_fbResult.P_MethodResult := ap_fbEventsExecute[0]^.M_Execute(_fbResult.P_MethodResult);
END_METHOD

METHOD PUBLIC M_ExecuteControl : HResult //needs to run all the time
VAR_INPUT
END_VAR
VAR
	loopCounter : DINT;
	currentState : E_PackMLStates;
END_VAR
_mapping();
currentState := state;
FOR loopCounter := 0 TO 20 BY 1 DO 
	CASE state OF
		E_PackMLStates.aborted:
			M_Aborted();
		E_PackMLStates.aborting:
			M_Aborting();
		E_PackMLStates.complete:
			stateMachineResult := M_Complete(stateMachineResult);
			IF stateMachineResult = MPM_FBResult.E_Result.S_OK THEN
				state := E_PackMLStates.complete;
			END_IF		
		E_PackMLStates.completing:	
			stateMachineResult := M_Completing(stateMachineResult);
			IF stateMachineResult = MPM_FBResult.E_Result.S_OK THEN
				state := E_PackMLStates.idle;
			END_IF					
		E_PackMLStates.execute:	
			stateMachineResult := M_Execute(stateMachineResult);	
			IF stateMachineResult = MPM_FBResult.E_Result.S_OK THEN
				state := E_PackMLStates.completing;
			END_IF			
		E_PackMLStates.held:	
			M_Held();	
		E_PackMLStates.holding:	
			M_Holding();		
		E_PackMLStates.idle:	
			stateMachineResult := M_Idle(stateMachineResult);		
			IF stateMachineResult = MPM_FBResult.E_Result.S_WORKING AND start = TRUE THEN
				stateMachineResult := MPM_FBResult.E_Result.S_OK;
				start := FALSE;
				state := E_PackMLStates.starting;
			END_IF	
		E_PackMLStates.starting:	
			stateMachineResult := M_Starting(stateMachineResult);
			IF stateMachineResult = MPM_FBResult.E_Result.S_OK THEN
				state := E_PackMLStates.execute;
			END_IF		
		E_PackMLStates.stopped:	
			M_Stopped();	
		E_PackMLStates.stopping:	
			M_Stopping();
		E_PackMLStates.suspdending:	
			M_Suspending();		
		E_PackMLStates.suspended:	
			M_Suspended();	
		E_PackMLStates.un_holding:	
			M_Un_Holding();			
		E_PackMLStates.un_suspsending:	
			M_Un_Suspending();					
	END_CASE
	
	IF currentState = state THEN // if state didnt change
	 	EXIT;
	ELSE // if state changed
		currentState := state;
	END_IF
	
END_FOR
END_METHOD

METHOD PUBLIC M_Held : HResult
VAR_INPUT
END_VAR
VAR_OUTPUT
	abort : BOOL;
	stop : BOOL;
END_VAR
END_METHOD

METHOD PUBLIC M_Holding : HResult
VAR_INPUT
END_VAR
VAR_OUTPUT
	abort : BOOL;
	stop : BOOL;
END_VAR
END_METHOD

METHOD PUBLIC M_Idle : HResult
VAR_INPUT
	lastResult : HResult;
END_VAR
VAR_OUTPUT
	abort : BOOL;
END_VAR
VAR_INST
	_fbResult : FB_ResultHelper_V2_1;	
	_lastResult : HRESULT;
	_state : POINTER TO DINT;
END_VAR
_state := ADR(state_idle);
IF _fbResult.M_MethodResult(M_Idle,lastResult,ADR(_lastResult)) = FALSE THEN
	RETURN;
END_IF

_fbResult.P_MethodResult := ap_fbEventsIdle[0]^.M_Execute(_fbResult.P_MethodResult);
END_METHOD

METHOD PUBLIC M_Resetting : HResult
VAR_INPUT
END_VAR
VAR_OUTPUT
	abort : BOOL;
	stop : BOOL;
END_VAR
END_METHOD

METHOD M_Starting : HResult
VAR_INPUT
	lastResult : HResult;
END_VAR
VAR_OUTPUT
	abort : BOOL;
END_VAR
VAR_INST
	_fbResult : FB_ResultHelper_V2_1;	
	_lastResult : HRESULT;
	_state : POINTER TO DINT;
END_VAR
_state := ADR(state_starting);
IF _fbResult.M_MethodResult(M_Starting,lastResult,ADR(_lastResult)) = FALSE THEN
	RETURN;
END_IF

IF _fbResult.P_MethodResult = E_Result.S_OK THEN
	_state^ := 0;
END_IF

_fbResult.P_MethodResult := ap_fbEventsStarting[0]^.M_Execute(_fbResult.P_MethodResult);
END_METHOD

METHOD PUBLIC M_Stopped : HResult
VAR_INPUT
	
END_VAR
VAR_OUTPUT
	abort : BOOL;
END_VAR
END_METHOD

METHOD PUBLIC M_Stopping : HResult
VAR_INPUT
END_VAR
VAR_OUTPUT
	abort : BOOL;
END_VAR
END_METHOD

METHOD PUBLIC M_Suspended : HREsult
VAR_INPUT
END_VAR
VAR_OUTPUT
	abort : BOOL;
	stop : BOOL;
END_VAR
END_METHOD

METHOD PUBLIC M_Suspending : HREsult
VAR_INPUT
END_VAR
VAR_OUTPUT
	abort : BOOL;
	stop : BOOL;
END_VAR
END_METHOD

METHOD PUBLIC M_Un_Holding : HREsult
VAR_INPUT
END_VAR
VAR_OUTPUT
	abort : BOOL;
	stop : BOOL;
END_VAR
END_METHOD

METHOD PUBLIC M_Un_Suspending : HREsult
VAR_INPUT
END_VAR
VAR_OUTPUT
	abort : BOOL;
	stop : BOOL;
END_VAR
END_METHOD

END_FUNCTION_BLOCK

// ---- FBs/Abstracts/FB_PackMLControl.TcPOU
(*
Standard way to control assests in system
*)
FUNCTION_BLOCK ABSTRACT FB_PackMLControl
VAR_INPUT
END_VAR
VAR_OUTPUT
END_VAR
VAR
	state_idle : DINT;
	state_starting : DINT;
	state_execute : DINT;	
	state_completing : DINT;			
	state_complete : DINT;		
	start : BOOL;
	complete : BOOL;
	stateMachineResult : HResult;
	packMLStop : BOOL;
END_VAR

METHOD PUBLIC ABSTRACT M_Aborted : HResult
VAR_INPUT
END_VAR
END_METHOD

METHOD PUBLIC ABSTRACT M_Aborting : HResult
VAR_INPUT
END_VAR
END_METHOD

METHOD PUBLIC ABSTRACT M_Complete : HResult
VAR_INPUT
	lastResult : HResult;
END_VAR
VAR_OUTPUT
	abort : BOOL;
END_VAR
END_METHOD

METHOD PUBLIC ABSTRACT M_Completing : HREsult
VAR_INPUT
	lastResult : HResult;
END_VAR
VAR_OUTPUT
	abort : BOOL;	
	stop : BOOL;
END_VAR
END_METHOD

METHOD PUBLIC ABSTRACT M_Execute : HResult
VAR_INPUT
	lastResult : HResult;
END_VAR
VAR_OUTPUT
	stop : BOOL;
	suspend : BOOL;
	hold : BOOL;
END_VAR
END_METHOD

METHOD PUBLIC ABSTRACT M_Held : HResult
VAR_INPUT
END_VAR
VAR_OUTPUT
	abort : BOOL;
	stop : BOOL;
END_VAR
END_METHOD

METHOD PUBLIC ABSTRACT M_Holding : HResult
VAR_INPUT
END_VAR
VAR_OUTPUT
	abort : BOOL;
	stop : BOOL;
END_VAR
END_METHOD

METHOD PUBLIC ABSTRACT M_Idle : HResult
VAR_INPUT
	lastResult : HResult;
END_VAR
VAR_OUTPUT
	abort : BOOL;
END_VAR
END_METHOD

METHOD PUBLIC ABSTRACT M_Resetting : HResult
VAR_INPUT
END_VAR
VAR_OUTPUT
	abort : BOOL;
	stop : BOOL;
END_VAR
END_METHOD

METHOD ABSTRACT M_Starting : HResult
VAR_INPUT
	lastResult : HResult;
END_VAR
VAR_OUTPUT
	abort : BOOL;
END_VAR
END_METHOD

METHOD PUBLIC ABSTRACT M_Stopped : HResult
VAR_INPUT
END_VAR
VAR_OUTPUT
	abort : BOOL;
END_VAR
END_METHOD

METHOD PUBLIC ABSTRACT M_Stopping : HResult
VAR_INPUT
END_VAR
VAR_OUTPUT
	abort : BOOL;
END_VAR
END_METHOD

METHOD PUBLIC ABSTRACT M_Suspended : HREsult
VAR_INPUT
END_VAR
VAR_OUTPUT
	abort : BOOL;
	stop : BOOL;
END_VAR
END_METHOD

METHOD PUBLIC ABSTRACT M_Suspending : HREsult
VAR_INPUT
END_VAR
VAR_OUTPUT
	abort : BOOL;
	stop : BOOL;
END_VAR
END_METHOD

METHOD PUBLIC ABSTRACT M_Un_Holding : HREsult
VAR_INPUT
END_VAR
VAR_OUTPUT
	abort : BOOL;
	stop : BOOL;
END_VAR
END_METHOD

METHOD PUBLIC ABSTRACT M_Un_Suspending : HREsult
VAR_INPUT
END_VAR
VAR_OUTPUT
	abort : BOOL;
	stop : BOOL;
END_VAR
END_METHOD

END_FUNCTION_BLOCK

// ---- FBs/FB_Kinenmatics.TcPOU
FUNCTION_BLOCK FB_Kinenmatics
VAR_INPUT
	intialVelocity : LREAL;
	jerkLimit : LREAL;
	accelLimit : LREAL;
	decelLimit : LREAL;
	velocityLimit : LREAL;
	positionDelta : LREAL;
	timeToComplete : LREAL;
	discriment : LREAL;
END_VAR
VAR_OUTPUT
	minTime : LREAL;
	velocityOutput : LREAL;
	accelOutput : LREAL;
	jerkOutput : LREAL;
	error : BOOL;
	errorMsg : STRING;	
END_VAR
VAR
	positionMid : LREAL;
	positionQuarter : LREAL;
	//Caculating max values for a Jerk limited move
	jerkMoveAccelMax : LREAL;
	jerkMoveTimeToMaxAccel : LREAL;
	jerkMoveVelocityAtMaxAccel : LREAL;	
	jerkMoveVelocityMax : LREAL;
	jerkMoveTimeToMaxVelocity : LREAL;
	jerkMoveTimeToCompleteMin : LREAL;
	jerkMoveJerkLimitForTargetTime : LREAL;
	
	accelMoveTimeToMaxAccel : LREAL;
	accelMoveMaxVelocity : LREAL;
	accelMoveTimeForAccelConstantMove : LREAL;
	accelMoveTimeToCompleteMove : LREAL;

	accelMoveNewMaxAccel: LREAL;

	accelVelocityMoveTimeToMaxVelocity : LREAL;	
	accelVelocityMoveTimeFromMaxVelocityToMidPoint : LREAL;	
	accelVelocityTimeToCompleteMove : LREAL;
	accelSegment : ARRAY [0..6] OF LREAL;
	velocitySegment	: ARRAY [0..6] OF LREAL;
	positionSegment : ARRAY [0..6] OF LREAL;
	
	a : LREAL;
	b : LREAL;
	c : LREAL;
	


END_VAR

IF positionDelta <= 0 OR timeToComplete <= 0 OR accelLimit <= 0 OR decelLimit <= 0 OR velocityLimit <= 0 OR jerkLimit <= 0 THEN
	RETURN;
END_IF

positionMid := positionDelta/2.0;
positionQuarter := positionDelta/4.0;

//Solve for t jerk limited equation positionMid = jerkLimit * t^3, 
//t = (positionMid/jerkLimit) ^(1/3) where t = 1/4 of the time to complete the move
jerkMoveTimeToMaxAccel := EXPT(positionMid/jerkLimit,1.0/3.0);
jerkMoveAccelMax := jerkLimit * jerkMoveTimeToMaxAccel;
jerkMoveVelocityAtMaxAccel := jerkMoveTimeToMaxAccel * jerkMoveAccelMax;
jerkMoveTimeToCompleteMin := jerkMoveTimeToMaxAccel * 4.0;

IF jerkMoveTimeToCompleteMin > timeToComplete THEN
	minTime := jerkMoveTimeToCompleteMin;
	errorMsg := 'Jerk limit too low';
	error := TRUE;			
	RETURN;
ELSE
	errorMsg := '';	
	error := FALSE;			
END_IF

IF (accelLimit < jerkMoveAccelMax) OR velocityLimit <= jerkMoveVelocityAtMaxAccel THEN
	//Caculate known values
	accelMoveTimeToMaxAccel := accelLimit/jerkLimit;
	positionSegment[0] := 1.0/6.0 * jerkLimit * EXPT(accelMoveTimeToMaxAccel,3.0);
	velocitySegment[0] := 0.5 * jerkLimit * EXPT(accelMoveTimeToMaxAccel,2.0) + intialVelocity;
	accelSegment[0] := jerkLimit*accelMoveTimeToMaxAccel;
	
	//set up quardatic formula 
	// 1/2*accelLimit*t^2 + (velocitySegment[0] + (accelLimit[0]*accelMoveTimeToMaxAccel)*t + (velocitySegment[0] * accelMoveTimeToMaxAccel)+accelSegment[0]*0.5*accelMoveTimeToMaxAccel^2
	a := 0.5 * accelSegment[0];
	b :=  velocitySegment[0] + accelSegment[0]*accelMoveTimeToMaxAccel;
	c := ((velocitySegment[0] * accelMoveTimeToMaxAccel)+accelSegment[0]*0.5*EXPT(accelMoveTimeToMaxAccel,2.0)) - positionMid;
	
	//Make sure discriment > 0 otherwise program will crash
	discriment := (EXPT(b,2.0) - 4.0 * a *c);
	IF discriment > 0 THEN
		//caculate min time
		accelMoveTimeForAccelConstantMove := (-b + EXPT(EXPT(b,2.0) -4.0 * a *c,0.5))/(2*a); //solve for quadtratic
		accelMoveTimeToCompleteMove := 2.0*(accelMoveTimeToMaxAccel * 2.0 + accelMoveTimeForAccelConstantMove); // This value is the fastest the machine can move with the accel limit
		accelMoveMaxVelocity := accelMoveTimeToCompleteMove/2*accelSegment[0]-EXPT(accelSegment[0],2.0)/jerkLimit;
		//end of caculate min time
		IF accelMoveMaxVelocity > velocityLimit THEN
			accelVelocityMoveTimeToMaxVelocity := velocityLimit/accelLimit + accelLimit/(jerkLimit);
			positionSegment[1] := velocitySegment[0]*(accelVelocityMoveTimeToMaxVelocity-2.0*accelMoveTimeToMaxAccel) + 0.5*accelLimit*EXPT((accelVelocityMoveTimeToMaxVelocity-2.0*accelMoveTimeToMaxAccel),2.0);
			velocitySegment[1] := velocitySegment[0] + accelLimit * (accelVelocityMoveTimeToMaxVelocity-2.0*accelMoveTimeToMaxAccel);
			positionSegment[2] := velocitySegment[1] * accelMoveTimeToMaxAccel +  0.5*accelLimit*EXPT((accelMoveTimeToMaxAccel),2.0) - 1.0/6.0 * jerkLimit * EXPT(accelMoveTimeToMaxAccel,3.0);
			//positionSegment[0] :=velocitySegment[0]*(accelVelocityMoveTimeToMaxVelocity-2.0*accelMoveTimeToMaxAccel);
			positionSegment[3] := positionMid - (positionSegment[0] + positionSegment[1] + positionSegment[2]);
			accelVelocityMoveTimeFromMaxVelocityToMidPoint := positionSegment[3]/velocityLimit;
			accelVelocityTimeToCompleteMove := 2.0*(accelVelocityMoveTimeToMaxVelocity + accelVelocityMoveTimeFromMaxVelocityToMidPoint);
			IF	accelVelocityTimeToCompleteMove < timeToComplete THEN
				errorMsg := '';		
				error := FALSE;						
				a := 1/jerkLimit;
				b := -(accelVelocityMoveTimeToMaxVelocity + timeToComplete - accelVelocityTimeToCompleteMove); //-timeToComplete/2.0; //
				c := velocityLimit;
				discriment := (EXPT(b,2.0) - 4.0 * a *c);
				IF discriment > 0 THEN
					minTime := accelVelocityTimeToCompleteMove;
					velocityOutput := velocityLimit;
					accelOutput := (-b - EXPT(EXPT(b,2.0) -4.0 * a *c,0.5))/(2*a);
					jerkOutput := jerkLimit; 
				END_IF	
			ELSIF accelVelocityTimeToCompleteMove > timeToComplete THEN
				minTime := accelVelocityTimeToCompleteMove;				
				errorMsg := 'velocity limit to low';	
				error := TRUE;		
				RETURN;	
			ELSIF accelVelocityTimeToCompleteMove = timeToComplete THEN
				minTime := accelVelocityTimeToCompleteMove;
				velocityOutput := velocityLimit;
				accelOutput := accelLimit;
				jerkOutput := jerkLimit; 			
			END_IF
		ELSIF accelMoveTimeToCompleteMove > timeToComplete THEN 
				minTime := accelMoveTimeToCompleteMove;			
			errorMsg := 'accel limit to low';
			error := TRUE;
			RETURN;
		ELSIF accelMoveTimeToCompleteMove < timeToComplete THEN
			minTime := accelMoveTimeToCompleteMove;
			error := FALSE;			
			errorMsg := '';	
			//Vmax = t*a-a^2/(2*j)
			//positionMid = Intergrate(Vmax) = timeToCompleteMove/(4.0 * jerkLimit)*a^2 + ((timeToCompleteMove/2)^2)/2; solve with quaddratic
			//timeToCompleteMove/(4.0 * jerkLimit)*a^2 + ((timeToCompleteMove/2)^2)/2 (*a??????) - positionMid
			a := -(timeToComplete/(4.0*jerkLimit));
			b := EXPT(timeToComplete/2.0,2.0)/2.0;
			c := -positionMid;			
			discriment := (EXPT(b,2.0) - 4.0 * a *c);
			IF discriment > 0 THEN
				accelOutput := (-b + EXPT(EXPT(b,2.0) -4.0 * a *c,0.5))/(2*a); //solve for quadtratic
			END_IF
			jerkOutput := jerkLimit;
			velocityOutput := velocityLimit;			
		ELSE
			error := FALSE;					
			errorMsg := '';	
		END_IF	
	END_IF
	//RETURN; // accel limited only
ELSIF accelLimit < jerkMoveAccelMax AND velocityLimit < jerkMoveVelocityAtMaxAccel THEN
	RETURN; // accel limited only and might be velocity limited
ELSIF accelLimit >= jerkMoveAccelMax AND velocityLimit >= jerkMoveVelocityAtMaxAccel THEN
	//jerkLimit = positionMid/(timeToComplete/4)^(3)
	minTime := jerkMoveTimeToCompleteMin;
	jerkMoveJerkLimitForTargetTime := positionMid/EXPT(timeToComplete/4,3.0);
	jerkOutput := jerkMoveJerkLimitForTargetTime;
	velocityOutput := velocityLimit;
	accelOutput := accelLimit;
	RETURN; // jerk limited
END_IF
	


// Max velocity in a jerk only limited move = positionMid = 1/2 * jerkLimit * t^2
// jerkMoveTimeToMaxVelocity := EXPT(positionMid*6/jerkLimit,1.0/3.0);
// jerkMoveVelocityMax := 1.0/2.0 * jerkLimit * EXPT(jerkMoveTimeToMaxVelocity,2);

METHOD M_CaculateTimePosToZeroVelocity : BOOL
VAR_INPUT
	intialVelocity : LREAL;
END_VAR
VAR_OUTPUT
	timeToZeroVelocity : LREAL;
	posAtZeroVelocity : LREAL;
	accelAtZero : LREAL;
END_VAR
IF jerkLimit > 0 THEN
	timeToZeroVelocity := EXPT(intialVelocity*2.0/jerkLimit,1.0/2.0);
	posAtZeroVelocity := intialVelocity*timeToZeroVelocity + 1.0/6.0 * jerkLimit * EXPT(timeToZeroVelocity,3.0);
	accelAtZero := 1.0/2.0 * jerkLimit * EXPT(timeToZeroVelocity,2.0);
END_IF
END_METHOD

END_FUNCTION_BLOCK

// ---- FUN/F_INIT_ST_AnyType.TcPOU
FUNCTION F_INIT_ST_AnyType : HResult
VAR_INPUT
	stAnyType : POINTER TO MPM_JsonParser.ST_AnyType_User;
END_VAR
VAR
	pBytePointer : POINTER TO BYTE;
END_VAR

IF stAnyType = 0 THEN
	F_INIT_ST_AnyType := MPM_FBResult.E_Result.S_FAILED;
	RETURN;
END_IF
IF stAnyType^.pvalue > 0 THEN
	F_INIT_ST_AnyType := MPM_FBResult.E_Result.S_FAILED;
	RETURN;
END_IF
CASE stAnyType^.typeclass OF
	MPM_JsonParser.E_TypeClassEx.TYPE_BOOL:
		stAnyType^.pvalue := __NEW(BOOL);	
		stAnyType^.diSize := SIZEOF(BOOL);
		F_INIT_ST_AnyType := MPM_FBResult.E_Result.S_OK;
	MPM_JsonParser.E_TypeClassEx.TYPE_BYTE:
		stAnyType^.pvalue := __NEW(BYTE);	
		stAnyType^.diSize := SIZEOF(BYTE);	
		F_INIT_ST_AnyType := MPM_FBResult.E_Result.S_OK;
	MPM_JsonParser.E_TypeClassEx.TYPE_LREAL:
		stAnyType^.pvalue := __NEW(LREAL);	
		stAnyType^.diSize := SIZEOF(LREAL);	
		F_INIT_ST_AnyType := MPM_FBResult.E_Result.S_OK;		
	MPM_JsonParser.E_TypeClassEx.TYPE_DINT:
		stAnyType^.pvalue := __NEW(DINT);	
		stAnyType^.diSize := SIZEOF(DINT);	
		F_INIT_ST_AnyType := MPM_FBResult.E_Result.S_OK;
	MPM_JsonParser.E_TypeClassEx.TYPE_LINT:
		stAnyType^.pvalue := __NEW(LINT);	
		stAnyType^.diSize := SIZEOF(LINT);
		F_INIT_ST_AnyType := MPM_FBResult.E_Result.S_OK;	
	MPM_JsonParser.E_TypeClassEx.TYPE_UDINT:
		stAnyType^.pvalue := __NEW(UDINT);	
		stAnyType^.diSize := SIZEOF(UDINT);
		F_INIT_ST_AnyType := MPM_FBResult.E_Result.S_OK;	
	MPM_JsonParser.E_TypeClassEx.TYPE_INT:
		stAnyType^.pvalue := __NEW(INT);	
		stAnyType^.diSize := SIZEOF(INT);
		F_INIT_ST_AnyType := MPM_FBResult.E_Result.S_OK;		
	MPM_JsonParser.E_TypeClassEx.TYPE_REAL:
		stAnyType^.pvalue := __NEW(REAL);	
		stAnyType^.diSize := SIZEOF(REAL);	
		F_INIT_ST_AnyType := MPM_FBResult.E_Result.S_OK;		
	MPM_JsonParser.E_TypeClassEx.TYPE_WORD:
		stAnyType^.pvalue := __NEW(WORD);	
		stAnyType^.diSize := SIZEOF(WORD);	
		F_INIT_ST_AnyType := MPM_FBResult.E_Result.S_OK;		
	ELSE
		F_INIT_ST_AnyType := MPM_FBResult.E_Result.S_FAILED;				
END_CASE

END_FUNCTION

// ---- FBs/Abstracts/FB_EventScheduler.TcPOU
(*
used to create event schedulers
*)

FUNCTION_BLOCK ABSTRACT FB_EventScheduler
VAR_INPUT
END_VAR
VAR_OUTPUT
END_VAR
VAR
END_VAR

gh

END_FUNCTION_BLOCK

// ---- FBs/Abstracts/FB_TimeEvents.TcPOU
(*
Standard way to set up time events in a system. might make an interface
*)
FUNCTION_BLOCK ABSTRACT FB_TimeEvents
VAR_INPUT
END_VAR
VAR_OUTPUT
END_VAR
VAR
END_VAR

END_FUNCTION_BLOCK

// ---- FBs/FB_EventArray.TcPOU
FUNCTION_BLOCK FB_EventArray
VAR_INPUT
END_VAR
VAR_OUTPUT
END_VAR
VAR
END_VAR

END_FUNCTION_BLOCK

// ---- FBs/IO_Mapping/FB_IOMappingJson.TcPOU
{attribute 'call_after_init'}
FUNCTION_BLOCK FB_IOMappingJson EXTENDS FB_JsonSchemaEx_OLD
VAR_OUTPUT
	P_sJsonid			: MPM_JsonParser.DUT_JsonSchema := (member := '_id', typeClass := E_TypeClassEx.TYPE_STRING,jsonValueRoot := jsonRoot);
	P_sJsonTimeStamp	: MPM_JsonParser.DUT_JsonSchema := (member := 'time_stamp', typeClass := E_TypeClassEx.TYPE_FILETIME,jsonValueRoot := jsonRoot);		
	P_sJsonValues		: MPM_JsonParser.DUT_JsonSchema := (member := 'values', typeClass := E_TypeClassEx.TYPE_JSON,jsonValueRoot := jsonRoot);
END_VAR
VAR
	jsonRoot : SJsonValue;	
END_VAR
VAR_OUTPUT
	//stIOMappingEthercat : ARRAY [0..NUM_OF_VARS] OF ST_IOMappingEthercatJson;	
END_VAR
VAR CONSTANT
	//NUM_OF_VARS : DINT := -1 + (SIZEOF(ST_Vars_IO_Mapping_Ethercat)/8) ;// 8 is SIZEOF(PVOID) (SIZEOF(ST_IO_Mapping)/SIZEOF(PVOID)) -1 won't complie
END_VAR

METHOD INTERNAL M_Add1 : UDINT
VAR_INPUT
	x : REFERENCE TO UDINT;
END_VAR
M_Add1 := x;
x := x + 1;
END_METHOD

METHOD PUBLIC  M_CreateSchemaJson : BOOL
VAR_IN_OUT
END_VAR
VAR
	json : sJsonValue;
END_VAR
jsonRoot := THIS^.NewDocument();
M_SetJsonSchema(jsonRoot,P_sJsonid);
//M_SetJsonSchema(P_sJsonid.jsonValue,P_sJsonRecipe);
M_SetJsonSchema(jsonRoot,P_sJsonValues);
M_SetJsonSchema(jsonRoot,P_sJsonTimeStamp);
END_METHOD

METHOD PUBLIC M_GetIOMappingJson : HRESULT
VAR_INPUT
	lastResult : HRESULT;
END_VAR
VAR_INPUT
	path : STRING;
END_VAR
VAR_IN_OUT
	stIOMapping : ARRAY [*] OF ST_IOMappingJson;
END_VAR
VAR_INPUT
	fbIOMapping : POINTER TO FB_IOMapping;	
END_VAR
VAR
	pJson : SJsonValue;
	upperBound : DINT; 
END_VAR
VAR_INST
	loadFile : BOOL;		
	x : UDINT;
	fileName : STRING;
	_state			: DINT;
	_fbResult		: FB_ResultHelper;	
	errorCode : HRESULT;
END_VAR
//THIS^.CopyDocument(aStringJson,SIZEOF(aStringJson));

IF _fbResult.M_MethodResult(M_GetIOMappingJson,lastResult) = FALSE THEN
	RETURN;
ELSE
	
	IF _fbResult.P_Result = E_Result.S_OK THEN //Reset
		_state := 0;	
		x := 0;
		fileName := path;
		loadFile := FALSE;
		THIS^.LoadDocumentFromFile(fileName,loadFile,hrErrorCode => errorCode);
		loadFile := TRUE;
	END_IF 
	
	_fbResult.P_Result := E_Result.S_WORKING; //Working	
	
	CASE _state OF
		0:	
			THIS^.LoadDocumentFromFile(fileName,loadFile,hrErrorCode => errorCode);
			IF loadFile = FALSE AND errorCode = 0 THEN
				_state := 1;
			ELSIF loadFile = FALSE AND errorCode < 0 THEN
				_fbResult.P_Result := E_Result.S_FAILED; //Working	
			END_IF		
		1:
			THIS^.M_PraseSchemaJson();
			upperBound := UPPER_BOUND(stIOMapping,1);
			FOR x := 0 TO upperBound BY 1 DO
				pJson := THIS^.FindMember(P_sJsonValues.jsonValue,stIOMapping[x].name);	
				IF pJson > 0 THEN
					THIS^.M_GetIOMappingJson_Values(pJson,ADR(stIOMapping[x]),fbIOMapping);
				END_IF	
			END_FOR
			_fbResult.P_Result := E_Result.S_OK; //Working
	END_CASE	

END_IF
END_METHOD

METHOD PROTECTED M_GetIOMappingJson_Values : HRESULT
VAR_INPUT
	pJson : SJsonValue;
	stIOMapping : POINTER TO ST_IOMappingJson;	
	fbIOMapping : POINTER TO FB_IOMapping;
END_VAR
VAR
END_VAR
THIS^.M_GetJsonMemberValue(pJson,'deviceNum',stIOMapping^.deviceNum);
THIS^.M_GetJsonMemberValue(pJson,'channel',stIOMapping^.channel);

THIS^.M_GetJsonMemberValue(pJson,'ethercatDeviceNum',stIOMapping^.ethercatDeviceNum);
THIS^.M_GetJsonMemberValue(pJson,'ioLinkDevice',stIOMapping^.ioLinkDevice);
THIS^.M_GetJsonMemberValue(pJson,'ioLinkSlaveChannel',stIOMapping^.ioLinkSlaveChannel);


IF stIOMapping^.deviceNum > 0 AND_THEN fbIOMapping^.ip.M_GetRef_PVOID((stIOMapping^.pAny.pvalue),stIOMapping^.deviceNum,stIOMapping^.channel) = MPM_FBResult.E_Result.S_FAILED THEN
	M_GetIOMappingJson_Values := E_Result.S_FAILED;
ELSIF stIOMapping^.ethercatDeviceNum > 0 AND_THEN fbIOMapping^.ip.M_GetRefIOLink_PVOID((stIOMapping^.pAny.pvalue),stIOMapping^.ethercatDeviceNum,stIOMapping^.ioLinkDevice,stIOMapping^.ioLinkSlaveChannel) = MPM_FBResult.E_Result.S_FAILED THEN
	M_GetIOMappingJson_Values :=  E_Result.S_FAILED;;	
END_IF

M_GetIOMappingJson_Values :=  E_Result.S_OK;
END_METHOD

METHOD PUBLIC  M_PraseSchemaJson : BOOL
VAR_INPUT
END_VAR
VAR
END_VAR
jsonRoot := THIS^.GetDocumentRoot();
IF jsonRoot > 0 THEN
	M_PraseJsonSchema(jsonRoot,P_sJsonid);
	//M_SetJsonSchema(P_sJsonid.jsonValue,P_sJsonRecipe);
	M_PraseJsonSchema(jsonRoot,P_sJsonValues);
	M_PraseJsonSchema(jsonRoot,P_sJsonTimeStamp);
END_IF
END_METHOD

METHOD PUBLIC M_SetIOMappingJson : HResult
VAR_INPUT
	lastResult : HRESULT;
END_VAR
VAR_INPUT
	path : STRING(255);
END_VAR
VAR_IN_OUT
	stIOMapping : ARRAY [*] OF ST_IOMappingJson;
END_VAR
VAR
	pJson : SJsonValue;
	upperBound : DINT; 
END_VAR
VAR_INST
	saveFile : BOOL;		
	x : UDINT;
	fileName : STRING(255);
	_state			: DINT;
	_fbResult		: FB_ResultHelper;	
	errorCode : HRESULT;
END_VAR
IF _fbResult.M_MethodResult(M_SetIOMappingJson,lastResult) = FALSE THEN
	RETURN;
ELSE
	
	IF _fbResult.P_Result = E_Result.S_OK THEN //Reset
		_state := 0;	
		x := 0;
		fileName := path;
		saveFile := FALSE;
		THIS^.SaveDocumentToFile(fileName,saveFile,hrErrorCode => errorCode);
		saveFile := TRUE;
	END_IF 
	
	_fbResult.P_Result := E_Result.S_WORKING; //Working	
	
	CASE _state OF
		0:	
			upperBound := UPPER_BOUND(stIOMapping,1);
			THIS^.M_CreateSchemaJson();
			
			FOR x := 0 TO upperBound BY 1 DO
				pJson := THIS^.M_SetJsonMember(P_sJsonValues.jsonValue,stIOMapping[x].name);		(* 3 Inches *)			
				THIS^.M_SetIOMappingJson_Values(pJson);
			END_FOR
			
			_state := 1;
		1:	
			THIS^.SaveDocumentToFile(fileName,saveFile,hrErrorCode => errorCode);
			IF saveFile = FALSE AND errorCode = 0 THEN
				_fbResult.P_Result := E_Result.S_OK; //Working	
			ELSIF saveFile = FALSE AND errorCode < 0 THEN
				_fbResult.P_Result := E_Result.S_FAILED; //Working	
			END_IF		
	END_CASE		
END_IF	



(*


*)
END_METHOD

METHOD PROTECTED M_SetIOMappingJson_Values : BOOL
VAR_INPUT
	pJson : SJsonValue;
END_VAR
VAR
	stIOMapping : ST_IOMappingJson;
END_VAR
THIS^.M_SetJsonMemberValue(pJson,'deviceNum',stIOMapping.deviceNum);
THIS^.M_SetJsonMemberValue(pJson,'channel',stIOMapping.channel);

THIS^.M_SetJsonMemberValue(pJson,'ethercatDeviceNum',stIOMapping.ethercatDeviceNum);
THIS^.M_SetJsonMemberValue(pJson,'ioLinkDevice',stIOMapping.ioLinkDevice);
THIS^.M_SetJsonMemberValue(pJson,'ioLinkSlaveChannel',stIOMapping.ioLinkSlaveChannel);
END_METHOD

END_FUNCTION_BLOCK

// ---- FBs/IO_Mapping/TcCom/FB_IOMapping.TcPOU
FUNCTION_BLOCK FB_IOMapping
VAR_OUTPUT
	ip : I_IOMapping;
END_VAR

VAR
	{attribute 'displaymode':='hex'}
	nObjId AT%I* : OTCID; 	// Instance configured to be retrieved
	iid : IID := TC_GLOBAL_IID_LIST.IID_I_IOMapping;
	

	
END_VAR

{attribute 'hide'}
METHOD FB_exit : BOOL
VAR_INPUT
	bInCopyCode : BOOL; // if TRUE, the exit method is called for exiting an instance that is copied afterwards (online change).
END_VAR
IF NOT bInCopyCode THEN // if not online change
	FW_SafeRelease(ADR(ip));
END_IF
END_METHOD

METHOD GetInterfacePointer : HRESULT
VAR
END_VAR
IF nObjID <> 0 THEN
	IF (ip = 0) THEN // only get interface pointer if it is not already existing
		GetInterfacePointer := FW_ObjMgr_GetObjectInstance(oid:=nObjID, iid:=iid, pipUnk:=ADR(ip));
	ELSE
		GetInterfacePointer := E_HRESULTAdsErr.EXISTS;
	END_IF
ELSE
	GetInterfacePointer := E_HRESULTAdsErr.INVALIDOBJID;
END_IF
END_METHOD

END_FUNCTION_BLOCK

// ---- FBs/JSON/FB_NCAxisJson.TcPOU
{attribute 'call_after_init'}
FUNCTION_BLOCK FB_NCAxisJson EXTENDS FB_JsonSchemaEx_OLD
VAR_INPUT
		
END_VAR
VAR_OUTPUT
	P_sJsonid			: MPM_JsonParser.DUT_JsonSchema := (member := '_id', typeClass := E_TypeClassEx.TYPE_STRING,jsonValueRoot := jsonRoot);
	P_sJsonTimeStamp	: MPM_JsonParser.DUT_JsonSchema := (member := 'time_stamp', typeClass := E_TypeClassEx.TYPE_FILETIME,jsonValueRoot := jsonRoot);		
	P_sJsonValues		: MPM_JsonParser.DUT_JsonSchema := (member := 'values', typeClass := E_TypeClassEx.TYPE_JSON,jsonValueRoot := jsonRoot);
END_VAR
VAR
	jsonRoot : SJsonValue;
	adsRead : ADSReadEX;
	saveTemplete : BOOL := FALSE;
	stAxisMappingJson : ARRAY [0..NUM_OF_VARS] OF  ST_AxisMapping;
END_VAR
VAR_OUTPUT
	//stIOMappingEthercat : ARRAY [0..NUM_OF_VARS] OF ST_IOMappingEthercatJson;	
END_VAR
VAR CONSTANT
	NUM_OF_VARS : DINT := 67 ;// 8 is SIZEOF(PVOID) (SIZEOF(ST_IO_Mapping)/SIZEOF(PVOID)) -1 won't complie
	INDEX_BASE : DINT :=  16384;
	PORT : UINT := 501;
END_VAR

METHOD PROTECTED _M_MapJsonValues : HRESULT
VAR_INPUT
	stAxisMappingJson : REFERENCE TO ST_AxisMapping;
	name : STRING;
	indexOffset : UDINT;
	pAny : ANY;
END_VAR
stAxisMappingJson.name := name;
stAxisMappingJson.indexOffset := indexOffset;
stAxisMappingJson.pAny.typeclass := TO_INT(pAny.TypeClass);
stAxisMappingJson.pAny.pvalue := pAny.pValue;
stAxisMappingJson.pAny.diSize := pAny.diSize;
END_METHOD

METHOD INTERNAL F_Add1 : UDINT
VAR_INPUT
	x : REFERENCE TO UDINT;
END_VAR
F_Add1 := x;
x := x + 1;
END_METHOD

METHOD PUBLIC  M_CreateSchemaJson : BOOL
VAR_IN_OUT
END_VAR
VAR
	
END_VAR
jsonRoot := THIS^.NewDocument();
M_SetJsonSchema(jsonRoot,P_sJsonid);
//M_SetJsonSchema(P_sJsonid.jsonValue,P_sJsonRecipe);
M_SetJsonSchema(jsonRoot,P_sJsonValues);
M_SetJsonSchema(jsonRoot,P_sJsonTimeStamp);
END_METHOD

METHOD PUBLIC M_GetAxisJson : HRESULT
VAR_INPUT
	lastResult : HRESULT;
END_VAR
VAR_INPUT
	path : STRING(255);
END_VAR
VAR_INPUT
	pAxisParamters : POINTER TO Tc2_MC2.ST_AxisParameterSet;
END_VAR
VAR_INST
	loadFile : BOOL;		
	x : UDINT;
	aStringJson : STRING(10000);
	fileName : STRING(255);
	_state			: DINT;
	_fbResult		: FB_ResultHelper;	
	errorCode : HRESULT;
END_VAR

VAR
	pJson : SJsonValue;
END_VAR
IF _fbResult.M_MethodResult(M_GetAxisJson,lastResult) = FALSE THEN
	RETURN;
ELSE

	IF _fbResult.P_Result = E_Result.S_OK THEN //Reset
		_state := 0;	
		x := 0;
		loadFile := FALSE;
		THIS^.LoadDocumentFromFile(fileName,loadFile,hrErrorCode => errorCode);
		loadFile := TRUE;
		errorCode := 0;
	END_IF 

	_fbResult.P_Result := E_Result.S_WORKING; //Working	
	
	CASE _state OF
		0:
			fileName := path;
			THIS^.LoadDocumentFromFile(fileName,loadFile,hrErrorCode => errorCode);
			IF loadFile = FALSE AND errorCode = 0 THEN
				_state := 1;	
			ELSIF loadFile = FALSE AND errorCode < 0 THEN
				_fbResult.P_Result := E_Result.S_FAILED; //Working	
			END_IF
		1:
			THIS^.M_PraseSchemaJson();
			FOR x := 0 TO NUM_OF_VARS BY 1 DO
				pJson := THIS^.FindMember(P_sJsonValues.jsonValue,stAxisMappingJson[x].name);	
				IF pJson > 0 THEN
					THIS^.M_GetAxisJson_Values(pJson,ADR(stAxisMappingJson[x]),pAxisParamters);
				END_IF	
			END_FOR	
			_fbResult.P_Result := E_Result.S_OK; //OK				
		END_CASE
END_IF
END_METHOD

METHOD PROTECTED M_GetAxisJson_Values : HResult
VAR_INPUT
	sJson : SJsonValue;
	stAxisMapping : POINTER TO ST_AxisMapping;
	pAxisParamters : POINTER TO Tc2_MC2.ST_AxisParameterSet;	
END_VAR

VAR
	pAny : MPM_JsonParser.ST_AnyType_User;	
END_VAR
pAny := stAxisMapping^.pAny;
pAny.pvalue := pAny.pvalue + pAxisParamters;
THIS^.M_GetJsonMemberValue_AnyType(sJson,'value',pAny);
END_METHOD

METHOD PUBLIC M_GetParametersFromAxis : HResult
VAR_INPUT
	lastResult : HRESULT;
	axisID : DINT;
	pAxisParamters : POINTER TO Tc2_Mc2.ST_AxisParameterSet;
END_VAR	


VAR_INST
	adsRead : ADSRead;	
	_state			: DINT;
	_fbResult		: FB_ResultHelper;
	x : DINT;
END_VAR
IF _fbResult.M_MethodResult(M_GetParametersFromAxis,lastResult) = FALSE THEN
	RETURN;
ELSE
	
	IF _fbResult.P_Result = E_Result.S_OK THEN //Reset
		_state := 0;	
		adsRead(READ := FALSE);
		x := 0;
	END_IF 
	
	_fbResult.P_Result := E_Result.S_WORKING; //Working	
	
	CASE _state OF
		0:
			adsRead.port := PORT;
			adsRead.IDXGRP := INDEX_BASE + axisID;
			adsRead.IDXOFFS :=stAxisMappingJson[x].indexOffset;
			adsRead.LEN := stAxisMappingJson[x].pAny.diSize;
			adsRead.DESTADDR := stAxisMappingJson[x].pAny.pvalue + pAxisParamters; //very important how this works
			adsRead(READ := TRUE);
			_state := 1;
		1:
			adsRead(READ := TRUE);
			IF adsRead.READ = TRUE AND adsRead.BUSY = FALSE AND adsRead.ERR = FALSE THEN
				IF x < NUM_OF_VARS THEN
					x := x + 1;
					adsRead(READ := FALSE);
					_state := 0;
				ELSIF x >= NUM_OF_VARS THEN
					_fbResult.P_Result := E_Result.S_OK;
				END_IF
			ELSIF adsRead.READ = TRUE AND adsRead.BUSY = FALSE AND adsRead.ERR = TRUE THEN
				ADSLOGSTR(msgCtrlMask := ADSLOG_MSGTYPE_ERROR,
					msgFmtStr := 'Error in %s',
					strArg := stAxisMappingJson[x].name);
				ADSLOGSTR(msgCtrlMask := ADSLOG_MSGTYPE_ERROR,
					msgFmtStr := 'ErrorID %s',
					strArg := TO_STRING(adsRead.ERRID));
				_fbResult.P_Result := E_Result.S_FAILED;	
			END_IF	
	END_CASE
END_IF
END_METHOD

METHOD PUBLIC M_MapJsonValues : HResult
VAR_INPUT
END_VAR

VAR
	x : UDINT;
	pAxisParamters : POINTER TO TC2_MC2.ST_AxisParameterSet;;	
END_VAR
(* AXIS: *)
_M_MapJsonValues(stAxisMappingJson[F_Add1(x)],'AxisId',16#1,pAxisParamters^.AxisId); // AxisId                      : DWORD; (* 0x00000001 *)
_M_MapJsonValues(stAxisMappingJson[F_Add1(x)],'sAxisName',16#2,pAxisParamters^.sAxisName);// sAxisName                   : STRING(31); (* 0x00000002 *)
_M_MapJsonValues(stAxisMappingJson[F_Add1(x)],'nAxisType',16#3,pAxisParamters^.nAxisType); // nAxisType                   : DWORD;      (* 0x00000003 *)
_M_MapJsonValues(stAxisMappingJson[F_Add1(x)],'bEnablePositionAreaControl',16#F,pAxisParamters^.bEnablePositionAreaControl);// bEnablePositionAreaControl  : WORD;       (* 0x0000000F *)
_M_MapJsonValues(stAxisMappingJson[F_Add1(x)],'fPositionAreaControlRange',16#10,pAxisParamters^.fPositionAreaControlRange);// fPositionAreaControlRange   : LREAL;      (* 0x00000010 *)
_M_MapJsonValues(stAxisMappingJson[F_Add1(x)],'bEnableMotionControl',16#11,pAxisParamters^.bEnableMotionControl);// bEnableMotionControl        : WORD;       (* 0x00000011 *)
_M_MapJsonValues(stAxisMappingJson[F_Add1(x)],'fMotionControlTime',16#12,pAxisParamters^.fMotionControlTime);// fMotionControlTime          : LREAL;      (* 0x00000012 *)
_M_MapJsonValues(stAxisMappingJson[F_Add1(x)],'bEnableLoop',16#13,pAxisParamters^.bEnableLoop);//   bEnableLoop                 : WORD;       (* 0x00000013 *)
_M_MapJsonValues(stAxisMappingJson[F_Add1(x)],'fLoopDistance',16#14,pAxisParamters^.fLoopDistance);// fLoopDistance               : LREAL;      (* 0x00000014 *)
_M_MapJsonValues(stAxisMappingJson[F_Add1(x)],'bEnableTargetPosControl',16#15,pAxisParamters^.bEnableTargetPosControl);// bEnableTargetPosControl     : WORD;       (* 0x00000015 *)
_M_MapJsonValues(stAxisMappingJson[F_Add1(x)],'fTargetPosControlRange',16#16,pAxisParamters^.fTargetPosControlRange);// fTargetPosControlRange      : LREAL;      (* 0x00000016 *)
_M_MapJsonValues(stAxisMappingJson[F_Add1(x)],'fTargetPosControlTime',16#17,pAxisParamters^.fTargetPosControlTime);// fTargetPosControlTime       : LREAL;      (* 0x00000017 *)
_M_MapJsonValues(stAxisMappingJson[F_Add1(x)],'fVeloMaximum',16#27,pAxisParamters^.fVeloMaximum);// fVeloMaximum                : LREAL;      (* 0x00000027 *)
_M_MapJsonValues(stAxisMappingJson[F_Add1(x)],'fMotionControlRange',16#28,pAxisParamters^.fMotionControlRange);// fMotionControlRange         : LREAL;      (* 0x00000028 *)
_M_MapJsonValues(stAxisMappingJson[F_Add1(x)],'bEnablePEHTimeControl',16#29,pAxisParamters^.bEnablePEHTimeControl);// bEnablePEHTimeControl       : WORD;       (* 0x00000029 *)
_M_MapJsonValues(stAxisMappingJson[F_Add1(x)],'fPEHControlTime',16#2A,pAxisParamters^.fPEHControlTime);// fPEHControlTime             : LREAL;      (* 0x0000002A *)
_M_MapJsonValues(stAxisMappingJson[F_Add1(x)],'bEnableBacklashCompensation',16#2B,pAxisParamters^.bEnableBacklashCompensation);// bEnableBacklashCompensation : WORD;       (* 0x0000002B *)
_M_MapJsonValues(stAxisMappingJson[F_Add1(x)],'fBacklash',16#2C,pAxisParamters^.fBacklash);// fBacklash                   : LREAL;      (* 0x0000002C *))
//_M_MapJsonValues(stAxisMappingJson[M_Add1(x)],'sAmsNetId',16#31,pAxisParamters^.sAmsNetId);// sAmsNetId : WORD;       (* 0x00000031 *)
//_M_MapJsonValues(stAxisMappingJson[M_Add1(x)],'nPort',16#31,pAxisParamters^.nPort);// nPort : WORD;       (* 0x00000031 *)*)
//_M_MapJsonValues(stAxisMappingJson[M_Add1(x)],'fDeceleration',16#102,pAxisParamters^.fDeceleration);//fDeceleration               : LREAL;      (* 0x00000101
//_M_MapJsonValues(stAxisMappingJson[M_Add1(x)],'nChnNo',16#31,pAxisParamters^.nChnNo);// nChnNo : WORD;       (* 0x00000031 *)
_M_MapJsonValues(stAxisMappingJson[F_Add1(x)],'fAcceleration',16#101,pAxisParamters^.fAcceleration);//fAcceleration               : LREAL;      (* 0x00000101 *)
_M_MapJsonValues(stAxisMappingJson[F_Add1(x)],'fDeceleration',16#102,pAxisParamters^.fDeceleration);//fDeceleration               : LREAL;      (* 0x00000102  *)
_M_MapJsonValues(stAxisMappingJson[F_Add1(x)],'fAccelerationMax',16#F1,pAxisParamters^.fAccelerationMax);//fAcceleration               : LREAL;      (* 0x00000101 *)
_M_MapJsonValues(stAxisMappingJson[F_Add1(x)],'fDecelerationMax',16#F2,pAxisParamters^.fDecelerationMax);//fDeceleration               : LREAL;      (* 0x00000102  *)
_M_MapJsonValues(stAxisMappingJson[F_Add1(x)],'fJerk',16#103,pAxisParamters^.fJerk);//fJerk                       : LREAL;      (* 0x00000103 *)
(* ENCODER: *)
_M_MapJsonValues(stAxisMappingJson[F_Add1(x)],'nEncId',16#10001,pAxisParamters^.nEncId);//nEncId                      : DWORD;      (* 0x00010001 *)
_M_MapJsonValues(stAxisMappingJson[F_Add1(x)],'sEncName',16#10002,pAxisParamters^.sEncName);//sEncName                    : STRING(31); (* 0x00010002 *)
_M_MapJsonValues(stAxisMappingJson[F_Add1(x)],'nEncType',16#10003,pAxisParamters^.nEncType);//nEncType                    : DWORD;      (* 0x00010003 *)
_M_MapJsonValues(stAxisMappingJson[F_Add1(x)],'fEncScaleFactorNumerator',16#10023,pAxisParamters^.fEncScaleFactorNumerator);//fEncScaleFactorNumerator    : LREAL;          (* 0x00010023 *)
_M_MapJsonValues(stAxisMappingJson[F_Add1(x)],'fEncScaleFactorDenominator',16#10024,pAxisParamters^.fEncScaleFactorDenominator);//fEncScaleFactorDenominator  : LREAL;          (* 0x00010024 *)
//_M_MapJsonValues(stAxisMappingJson[M_Add1(x)],'fEncScaleFactorInternal',16#10024,pAxisParamters^.fEncScaleFactorInternal);//fEncScaleFactorDenominator  : LREAL;          (* 0x00010024 *)
_M_MapJsonValues(stAxisMappingJson[F_Add1(x)],'fEncOffset',16#10007,pAxisParamters^.fEncOffset);//fEncOffset                  : LREAL;      (* 0x00010007 *)
_M_MapJsonValues(stAxisMappingJson[F_Add1(x)],'bEncIsInverse',16#10008,pAxisParamters^.bEncIsInverse);//bEncIsInverse               : WORD;       (* 0x00010008 *)
_M_MapJsonValues(stAxisMappingJson[F_Add1(x)],'fEncModuloFactor',16#10009,pAxisParamters^.fEncModuloFactor);//fEncModuloFactor            : LREAL;      (* 0x00010009 *)
_M_MapJsonValues(stAxisMappingJson[F_Add1(x)],'nEncMode',16#1000A,pAxisParamters^.nEncMode);//nEncMode                    : DWORD;      (* 0x0001000A *)
_M_MapJsonValues(stAxisMappingJson[F_Add1(x)],'bEncEnableSoftEndMinControl',16#1000B,pAxisParamters^.bEncEnableSoftEndMinControl);//bEncEnableSoftEndMinControl : WORD;       (* 0x0001000B *)
_M_MapJsonValues(stAxisMappingJson[F_Add1(x)],'bEncEnableSoftEndMaxControl',16#1000C,pAxisParamters^.bEncEnableSoftEndMaxControl);//bEncEnableSoftEndMaxControl : WORD;       (* 0x0001000C *)
_M_MapJsonValues(stAxisMappingJson[F_Add1(x)],'fEncSoftEndMin',16#1000D,pAxisParamters^.fEncSoftEndMin);//fEncSoftEndMin              : LREAL;      (* 0x0001000D *)
_M_MapJsonValues(stAxisMappingJson[F_Add1(x)],'fEncSoftEndMax',16#1000E,pAxisParamters^.fEncSoftEndMax);//fEncSoftEndMax              : LREAL;      (* 0x0001000E *)
_M_MapJsonValues(stAxisMappingJson[F_Add1(x)],'nEncMaxIncrement',16#10015,pAxisParamters^.nEncMaxIncrement);//nEncMaxIncrement            : DWORD;      (* 0x00010015 *)
_M_MapJsonValues(stAxisMappingJson[F_Add1(x)],'bEncEnablePosCorrection',16#10016,pAxisParamters^.bEncEnablePosCorrection);//bEncEnablePosCorrection     : WORD;       (* 0x00010016 *)
_M_MapJsonValues(stAxisMappingJson[F_Add1(x)],'fEncPosCorrectionFilterTime',16#10017,pAxisParamters^.fEncPosCorrectionFilterTime);//fEncPosCorrectionFilterTime : LREAL;      (* 0x00010017 *)
//_M_MapJsonValues(stAxisMappingJson[M_Add1(x)],'nEncReferenceSystem',16#100019,pAxisParamters^.nEncReferenceSystem);//nEncReferenceSystem         : DWORD;          (* 0x00010019 *)
(* CONTROLLER: *)
_M_MapJsonValues(stAxisMappingJson[F_Add1(x)],'nCtrlId',16#20001,pAxisParamters^.nCtrlId);//nCtrlId                     : DWORD;      (* 0x00020001 *)
_M_MapJsonValues(stAxisMappingJson[F_Add1(x)],'sCtrlName',16#20002,pAxisParamters^.sCtrlName);//sCtrlName                   : STRING(31); (* 0x00020002 *)
_M_MapJsonValues(stAxisMappingJson[F_Add1(x)],'nCtrlType',16#20003,pAxisParamters^.nCtrlType);//nCtrlType                   : DWORD;      (* 0x00020003 *)
_M_MapJsonValues(stAxisMappingJson[F_Add1(x)],'bCtrlEnablePosDiffControl',16#20010,pAxisParamters^.bCtrlEnablePosDiffControl);//bCtrlEnablePosDiffControl   : WORD;       (* 0x00020010 *)
_M_MapJsonValues(stAxisMappingJson[F_Add1(x)],'bCtrlEnableVeloDiffControl',16#20011,pAxisParamters^.bCtrlEnableVeloDiffControl);//bCtrlEnableVeloDiffControl  : WORD;       (* 0x00020011 *)
_M_MapJsonValues(stAxisMappingJson[F_Add1(x)],'fCtrlPosDiffMax',16#20012,pAxisParamters^.fCtrlPosDiffMax);//fCtrlPosDiffMax             : LREAL;      (* 0x00020012 *)
_M_MapJsonValues(stAxisMappingJson[F_Add1(x)],'fCtrlPosDiffMaxTime',16#20012,pAxisParamters^.fCtrlPosDiffMaxTime);//fCtrlPosDiffMaxTime         : LREAL;      (* 0x00020013 *)
_M_MapJsonValues(stAxisMappingJson[F_Add1(x)],'fCtrlPosKp',16#20102,pAxisParamters^.fCtrlPosKp);//fCtrlPosKp                  : LREAL;      (* 0x00020102 *)
_M_MapJsonValues(stAxisMappingJson[F_Add1(x)],'fCtrlPosTn',16#20103,pAxisParamters^.fCtrlPosTn);//fCtrlPosTn                  : LREAL;      (* 0x00020103 *)
_M_MapJsonValues(stAxisMappingJson[F_Add1(x)],'fCtrlPosTv',16#20104,pAxisParamters^.fCtrlPosTv);//fCtrlPosTv                  : LREAL;      (* 0x00020104 *)
_M_MapJsonValues(stAxisMappingJson[F_Add1(x)],'fCtrlPosTd',16#20105,pAxisParamters^.fCtrlPosTd);//fCtrlPosTd                  : LREAL;      (* 0x00020105 *)
_M_MapJsonValues(stAxisMappingJson[F_Add1(x)],'fCtrlPosExtKp',16#20106,pAxisParamters^.fCtrlPosExtKp);//fCtrlPosExtKp               : LREAL;      (* 0x00020106 *)
_M_MapJsonValues(stAxisMappingJson[F_Add1(x)],'fCtrlPosExtVelo',16#20107,pAxisParamters^.fCtrlPosExtVelo);//fCtrlPosExtVelo             : LREAL;      (* 0x00020107 *)
_M_MapJsonValues(stAxisMappingJson[F_Add1(x)],'fCtrlAccKa',16#20108,pAxisParamters^.fCtrlAccKa);//fCtrlAccKa                  : LREAL;      (* 0x00020108 *)
(* DRIVE: *)
_M_MapJsonValues(stAxisMappingJson[F_Add1(x)],'nDriveId',16#30001,pAxisParamters^.nDriveId);//nDriveId                    : DWORD;      (* 0x00030001 *)
_M_MapJsonValues(stAxisMappingJson[F_Add1(x)],'sDriveName',16#30002,pAxisParamters^.sDriveName);//sDriveName                  : STRING(31); (* 0x00030002 *)
_M_MapJsonValues(stAxisMappingJson[F_Add1(x)],'nDriveType',16#30003,pAxisParamters^.nDriveType);//nDriveType                  : DWORD;      (* 0x00030003 *)
_M_MapJsonValues(stAxisMappingJson[F_Add1(x)],'bDriveIsInverse',16#30006,pAxisParamters^.bDriveIsInverse);//bDriveIsInverse             : WORD;       (* 0x00030006 *)
_M_MapJsonValues(stAxisMappingJson[F_Add1(x)],'fDriveVeloReferenz',16#30101,pAxisParamters^.fDriveVeloReferenz);//fDriveVeloReferenz          : LREAL;      (* 0x00030101 *)
_M_MapJsonValues(stAxisMappingJson[F_Add1(x)],'fDriveOutputReferenz',16#30102,pAxisParamters^.fDriveOutputReferenz);//fDriveOutputReferenz        : LREAL;      (* 0x00030102 *)
_M_MapJsonValues(stAxisMappingJson[F_Add1(x)],'fDriveOutputScalingAcc',16#3010A,pAxisParamters^.fDriveOutputScalingAcc);//fDriveOutputScalingAcc      : LREAL;        (* 0x0003000A *)
_M_MapJsonValues(stAxisMappingJson[F_Add1(x)],'fDriveOutputScalingTorque',16#3010C,pAxisParamters^.fDriveOutputScalingTorque);//fDriveOutputScalingTorque   : LREAL;        (* 0x0003000B *)
_M_MapJsonValues(stAxisMappingJson[F_Add1(x)],'fDriveInputScalingTorque',16#30031,pAxisParamters^.fDriveInputScalingTorque);//fDriveInputScalingTorque    : LREAL;        (* 0x00030031 *)
_M_MapJsonValues(stAxisMappingJson[F_Add1(x)],'fDriveInputFiltertimeTorque',16#30032,pAxisParamters^.fDriveInputFiltertimeTorque);//fDriveInputFiltertimeTorque : LREAL;        (* 0x00030032 *)
_M_MapJsonValues(stAxisMappingJson[F_Add1(x)],'fDriveInputFiltertimeTorqueDerivative',16#30033,pAxisParamters^.fDriveInputFiltertimeTorqueDerivative);//fDriveInputFiltertimeTorqueDerivative: LREAL;(* 0x00030033 *)
(* miscellaneous *)
//_M_MapJsonValues(stAxisMappingJson[M_Add1(x)],'fAxisCycleTime',16#00000004,pAxisParamters^.fAxisCycleTime);//fAxisCycleTime              : LREAL;      (* 0x00000004 *) (* available from Tc 2.11 R2 *)
(* 17.05.11: parameter extension *)
_M_MapJsonValues(stAxisMappingJson[F_Add1(x)],'fRefVeloSearch',16#00000006,pAxisParamters^.fRefVeloSearch);//fRefVeloSearch              : LREAL;      (* 0x00000006 calibration velo (TO plc cam) *)
_M_MapJsonValues(stAxisMappingJson[F_Add1(x)],'fRefVeloSync',16#00000007,pAxisParamters^.fRefVeloSync);// fRefVeloSync                : LREAL;      (* 0x00000007 calibration velo (off plc cam) *)
_M_MapJsonValues(stAxisMappingJson[F_Add1(x)],'fVeloSlowManual',16#00000008,pAxisParamters^.fVeloSlowManual);//fVeloSlowManual             : LREAL;      (* 0x00000008 manual velocity (slow) *)
_M_MapJsonValues(stAxisMappingJson[F_Add1(x)],'fVeloFastManual',16#00000009,pAxisParamters^.fVeloFastManual);//fVeloFastManual             : LREAL;      (* 0x00000009 manual velocity (fast) *)
(* ENCODER (incremental): *)
//_M_MapJsonValues(stAxisMappingJson[M_Add1(x)],'bEncRefSearchInverse',16#10101,pAxisParamters^.bEncRefSearchInverse);//bEncRefSearchInverse        : UINT;       (* 0x00010101 *)
//_M_MapJsonValues(stAxisMappingJson[M_Add1(x)],'bEncRefSyncInverse',16#10102,pAxisParamters^.bEncRefSyncInverse);//bEncRefSyncInverse          : UINT;       (* 0x00010102 *)
//_M_MapJsonValues(stAxisMappingJson[M_Add1(x)],'nEncRefMode',16#10107,pAxisParamters^.nEncRefMode);//nEncRefMode                 : UDINT;      (* 0x00010107 *)
//_M_MapJsonValues(stAxisMappingJson[M_Add1(x)],'fEncRefPosition',16#00010103,pAxisParamters^.fEncRefPosition);//fEncRefPosition             : LREAL;      (* 0x00010103 *)
END_METHOD

METHOD PUBLIC  M_PraseSchemaJson : BOOL
VAR_INPUT
END_VAR
VAR
END_VAR
jsonRoot := THIS^.GetDocumentRoot();
IF jsonRoot > 0 THEN
	M_PraseJsonSchema(jsonRoot,P_sJsonid);
	//M_SetJsonSchema(P_sJsonid.jsonValue,P_sJsonRecipe);
	M_PraseJsonSchema(jsonRoot,P_sJsonValues);
	M_PraseJsonSchema(jsonRoot,P_sJsonTimeStamp);
END_IF
END_METHOD

METHOD PUBLIC M_SetAxisJson : HResult
VAR_INPUT
	lastResult : HRESULT;
END_VAR
VAR_INPUT
	path : STRING(255);
END_VAR
VAR_INPUT
	pAxisParamters : POINTER TO Tc2_MC2.ST_AxisParameterSet;
END_VAR

VAR
	pJson : SJsonValue;
END_VAR

VAR_INST
	saveFile : BOOL;		
	x : UDINT;
	aStringJson : STRING(10000);
	fileName : STRING(255);
	_state			: DINT;
	_fbResult		: FB_ResultHelper;	
	errorCode : HRESULT;
END_VAR
IF _fbResult.M_MethodResult(M_SetAxisJson,lastResult) = FALSE THEN
	RETURN;
ELSE

	IF _fbResult.P_Result = E_Result.S_OK THEN //Reset
		_state := 0;	
		x := 0;
		saveFile := FALSE;
		errorCode := 0;
		THIS^.SaveDocumentToFile(fileName,saveFile,hrErrorCode => errorCode);
		saveFile := TRUE;
		fileName := path;
	END_IF 

	_fbResult.P_Result := E_Result.S_WORKING; //Working	
	
	CASE _state OF
		0:
			THIS^.M_CreateSchemaJson();
			FOR x := 0 TO NUM_OF_VARS BY 1 DO
				pJson := THIS^.M_SetJsonMember(P_sJsonValues.jsonValue,stAxisMappingJson[x].name);		(* 3 Inches *)			
				THIS^.M_SetAxisJson_Values(pJson,ADR(stAxisMappingJson[x]),(pAxisParamters));
			END_FOR
			_state := 1;
		1:		
			THIS^.SaveDocumentToFile(fileName,saveFile,hrErrorCode => errorCode);
			IF saveFile = FALSE AND errorCode = 0 THEN
				_fbResult.P_Result := E_Result.S_OK; //Working	
			ELSIF saveFile = FALSE AND errorCode < 0 THEN
				_fbResult.P_Result := E_Result.S_FAILED; //Working	
			END_IF		
	END_CASE	
	
	
END_IF
END_METHOD

METHOD PROTECTED M_SetAxisJson_Values : HResult
VAR_INPUT
	sJson : SJsonValue;
	stAxisMapping : POINTER TO ST_AxisMapping;
	pAxisParamters : POINTER TO Tc2_MC2.ST_AxisParameterSet;
END_VAR
VAR
	pAny : MPM_JsonParser.ST_AnyType_User;	
END_VAR
pAny := stAxisMapping^.pAny; //copy so can be modified 
pAny.pvalue := pAny.pvalue + pAxisParamters; //very important how this works
THIS^.M_SetJsonMemberValue_AnyType(sJson,'value',pAny);
THIS^.M_SetJsonMemberValue(sJson,'indexOffset',stAxisMapping^.indexOffset);
END_METHOD

METHOD PUBLIC M_SetParametersToAxis : HRESULT
VAR_INPUT
	lastResult : HRESULT;
	axisID : DINT;
	pAxisParamters : POINTER TO Tc2_Mc2.ST_AxisParameterSet;
END_VAR
VAR_INST
	adsWrite : ADSWRITE;	
	_state			: DINT;
	_fbResult		: FB_ResultHelper;
	x : DINT;
END_VAR
IF _fbResult.M_MethodResult(M_SetParametersToAxis,lastResult) = FALSE THEN
	RETURN;
ELSE

	IF _fbResult.P_Result = E_Result.S_OK THEN //Reset
		_state := 0;	
		adsWrite(WRITE := FALSE);
		x := 0;
	END_IF 
		
	_fbResult.P_Result := E_Result.S_WORKING; //Working	
	
	CASE _state OF
		0:
			adsWrite.port := PORT;
			adsWrite.IDXGRP := INDEX_BASE + axisID;
			adsWrite.IDXOFFS :=stAxisMappingJson[x].indexOffset;
			adsWrite.LEN := (stAxisMappingJson[x].pAny.diSize);
			adsWrite.SRCADDR := (stAxisMappingJson[x].pAny.pvalue + pAxisParamters);
			adsWrite(WRITE := TRUE);
			_state := 1;
		1:
			adsWrite(WRITE := TRUE);
			IF adsWrite.WRITE = TRUE AND adsWrite.BUSY = FALSE AND adsWrite.ERR = FALSE THEN
				IF x < NUM_OF_VARS THEN
					x := x + 1;
					adsWrite(WRITE := FALSE);
					_state := 0;
				ELSIF x >= NUM_OF_VARS THEN
					_fbResult.P_Result := E_Result.S_OK;
				END_IF
			ELSIF adsWrite.WRITE = TRUE AND adsWrite.BUSY = FALSE AND adsWrite.ERR = TRUE THEN
				ADSLOGSTR(msgCtrlMask := ADSLOG_MSGTYPE_ERROR,
					msgFmtStr := 'Error in %s',
					strArg := stAxisMappingJson[x].name);
				ADSLOGSTR(msgCtrlMask := ADSLOG_MSGTYPE_ERROR,
					msgFmtStr := 'ErrorID %s',
					strArg := TO_STRING(adsWrite.ERRID));
				IF x < NUM_OF_VARS THEN
					x := x + 1;
					adsWrite(WRITE := FALSE);
					_state := 0;
				ELSIF x >= NUM_OF_VARS THEN
					_fbResult.P_Result := E_Result.S_OK;
				END_IF
			END_IF	
	END_CASE
	
END_IF
END_METHOD

END_FUNCTION_BLOCK

// ---- FBs/Main/FB_JsonFile.TcPOU
(*
used to write all values to and from json files. Will add to lib later
*)

FUNCTION_BLOCK ABSTRACT FB_JsonFile EXTENDS FB_JsonSchemaEx_OLD
VAR_INPUT
END_VAR
VAR_OUTPUT
END_VAR
VAR
END_VAR

END_FUNCTION_BLOCK

// ---- FBs/Main/FB_Squeegee.TcPOU
FUNCTION_BLOCK FB_Squeegee EXTENDS FB_ConfigBase
VAR_INPUT
END_VAR
VAR_OUTPUT
END_VAR
//axis
VAR
	axis : Tc2_MC2.AXIS_REF;	
	stAxisParameterSet : Tc2_MC2.ST_AxisParameterSet;  
	fbAxisControl : FB_AxisControl(axis);	
	fbKinenmatics2 : FB_Kinenmatics_V2;		
END_VAR
//recipe
VAR
	passThru : LREAL;	
	timeToClose : LREAL := 0.1; //100ms
	timeToOpen : LREAL := 0.1;	//100ms
END_VAR
//IO
VAR
	bagPosition AT %I* : LREAL;
	pullBeltVelocity AT %I*  : LREAL;
	pullBeltAccel AT %I*  : LREAL;
	pullBeltDecel AT %I* : LREAL;
END_VAR

METHOD _F_Axis : HRESULT
VAR_IN_OUT
	a_pstAxisParameterSet : POINTER TO Tc2_MC2.ST_AxisParameterSet; //pointer to array
	pstAxisMapping : UDINT;
END_VAR
stAxisParameterSet.AxisId := axis.NcToPlc.AxisId;
a_pstAxisParameterSet := ADR(stAxisParameterSet);
pstAxisMapping := SIZEOF(stAxisParameterSet);

_F_Axis := MPM_FBResult.E_Result.S_OK;
END_METHOD

METHOD PROTECTED  _F_IO : HResult
VAR_IN_OUT
	a_pstIOMappingJson : POINTER TO ST_IOMappingJson; //pointer to array
	ustIOMappingJson : UDINT; 		
END_VAR
VAR_INST
	stIOMappingJson : ARRAY [0..1] OF ST_IOMappingJson;
END_VAR
VAR
	x : DINT;
END_VAR
//	ioVar : POINTER TO BOOL;
//	ioVar2 : POINTER TO REAL;
//F_Map_ST_IOMappingJson(ADR(a_pstIOMappingJson[F_Add1(x)]),'lowLevelSensor',ADR(lowLevelSensor));
//F_Map_ST_IOMappingJson(ADR(a_pstIOMappingJson[F_Add1(x)]),'HighLevelSensor',ADR(HighLevelSensor));

//a_pstIOMappingJson := ADR(stIOMappingJson);
//ustIOMappingJson := SIZEOF(stIOMappingJson);




_F_IO := MPM_FBResult.E_Result.S_OK;
END_METHOD

(*
return the list of vars that want to be saved and loaded 
*)

METHOD PROTECTED  _F_Recipe : HResult
VAR_IN_OUT
	a_pstAnyTypeUser : POINTER TO MPM_JsonParser.ST_AnyType_User; //pointer to array
	uAnyTypeUser : UDINT; //size of array	
END_VAR
VAR_OUTPUT
END_VAR
VAR
	x : DINT;
END_VAR
VAR_INST
	a_stAnyTypeUser : ARRAY [0..0] OF MPM_JsonParser.ST_AnyType_User;
END_VAR
MPM_JsonParser.F_Map_ST_AnyType_User('volume',passThru,a_stAnyTypeUser[F_Add1(x)]);
//MPM_JsonParser.F_Map_ST_AnyType_User('timeToDispense',timeToDispense,a_stAnyTypeUser[F_Add1(x)]);


a_pstAnyTypeUser := ADR(a_stAnyTypeUser);
uAnyTypeUser := SIZEOF(a_stAnyTypeUser);

_F_Recipe := MPM_FBResult.E_Result.S_OK;
END_METHOD

METHOD PROTECTED _F_System : HResult
VAR_IN_OUT
	a_pstAnyTypeUser : POINTER TO MPM_JsonParser.ST_AnyType_User; //pointer to array
	uAnyTypeUser : UDINT; //size of array	
END_VAR
VAR_INST
	a_stAnyTypeUser : ARRAY [0..0] OF MPM_JsonParser.ST_AnyType_User;
END_VAR
VAR
	x : DINT;
END_VAR
//MPM_JsonParser.F_Map_ST_AnyType_User('volumePerRotation',volumePerRotation,a_stAnyTypeUser[F_Add1(x)]);


//a_pstAnyTypeUser := ADR(a_stAnyTypeUser);
//uAnyTypeUser := SIZEOF(a_stAnyTypeUser);

_F_System := MPM_FBResult.E_Result.S_OK;
END_METHOD

METHOD PUBLIC  M_Events : HResult
VAR_INPUT
	lastResult : HResult;
	eventID : DINT;
END_VAR
VAR_INST
	_fbResult : FB_ResultHelper_V2_1;
	_lastResult : HResult;
	openValve_Result : HRESULT;
	closeValve_Result : HRESULT;
	enablePump_Result : HRESULT;
	homeDirect_Result : HRESULT; 
	moveABS_Result : HRESULT; 	
	moveInter_Result : HRESULT; 		
	moveVelocity_Result : HRESULT; 		
	halt_Result : HRESULT;
END_VAR
VAR 
	HomingMode : Tc2_MC2.MC_HomingMode;
	OptionsHomeing : Tc2_MC2.ST_HomingOptions;
	BufferMode : Tc2_MC2.MC_BufferMode;
	OptionsPower : Tc2_MC2.ST_PowerOptions;	
	Options : Tc2_MC2.ST_MoveOptions;		
END_VAR

VAR_INST
	executeDyn : BOOL;
	VelocityDyn : LREAL := 10; 
END_VAR
CASE eventID OF 
	3: //enable pump
		IF _fbResult.M_MethodResult(M_Events,lastResult,ADR(enablePump_Result)) = FALSE THEN
			RETURN;
		END_IF	
		_fbResult.P_MethodResult := fbAxisControl.MC_Power(_fbResult.P_MethodResult,TRUE,TRUE,TRUE,100.0,BufferMode,OptionsPower);
	4: //Home Pump
		IF _fbResult.M_MethodResult(M_Events,lastResult,ADR(homeDirect_Result)) = FALSE THEN
			RETURN;
		END_IF			
		HomingMode := Tc2_MC2.MC_HomingMode.MC_Direct; 
		_fbResult.P_MethodResult := fbAxisControl.MC_Home(_fbResult.P_MethodResult,0.0,HomingMode,BufferMode,OptionsHomeing);
	6: //halt pump
		IF _fbResult.M_MethodResult(M_Events,lastResult,ADR(halt_Result)) = FALSE THEN
			RETURN;
		END_IF			
		_fbResult.P_MethodResult := fbAxisControl.MC_Halt(_fbResult.P_MethodResult,
			1000.0,
			1000.0);				
	8: //pump_intermeate
	fbKinenmatics2.jerkLimit := 100000;
	fbKinenmatics2.accelLimit := 15000.0;	
	fbKinenmatics2.decelLimit := 15000.0;	
	fbKinenmatics2.velocityLimit := 2500;	
	fbKinenmatics2.positionDelta := passThru;		
	fbKinenmatics2.timeToComplete := timeToDispense;
	fbKinenmatics2();
	IF _fbResult.M_MethodResult(M_Events,lastResult,ADR(moveInter_Result)) = FALSE THEN
			RETURN;
		END_IF		
		_fbResult.P_MethodResult := fbAxisControl.MC_MoveRelative(
			_fbResult.P_MethodResult,
			volume,
			fbKinenmatics2.velocityOutput,
			fbKinenmatics2.accelOutput,			
			fbKinenmatics2.decelLimit,		
			fbKinenmatics2.jerkOutput,		
			BufferMode,
			Options);			
END_CASE
END_METHOD

METHOD PUBLIC M_Execute : HRESULT
VAR_INPUT
END_VAR
fbAxisControl.M_Execute();
END_METHOD

END_FUNCTION_BLOCK
